FUNCTION FC_GetEpochTime : ULINT	// Returns the current EPOCH time

FC_GetEpochTime := IING.epochtime;

END_FUNCTION

(* stored: Version 1.1.0.1, ProductVersion 3.1.4026.18
   POU FC_GetEpochTime: Id {14513e43-2c1f-48e3-8165-5a5e0f64d099}, SpecialFunc None *)
